FUNCTION F_Change_Param : BOOL
VAR_INPUT
	IObject: I_Object;
	value: STRING;
END_VAR
VAR
	_IParam: I_Param;
	_interface_match: BOOL;
END_VAR

//Used to safely change param of unknown object. If object doesn't contain I_Param
//or if it is 0 then it won't work.

_interface_match := __QUERYINTERFACE(IObject, _IParam);
IF _interface_match THEN
	_IParam.Change_Param(value);
END_IF

F_Change_Param := _interface_match;

END_FUNCTION

(* stored: Version 1.1.0.1, ProductVersion 3.1.4024.12
   POU F_Change_Param: Id {1b59bbb4-5d51-4efd-9d96-47d8a2742135}, SpecialFunc None *)
